{attribute 'qualified_only' := ''}
{attribute 'strict' := ''}
TYPE eFirmerVendorEvent2 :
(
	eNoInfo := 0,
	ePowerLimitationForHighTemperature := 1,
	ePowerLimitationForHighDCVoltage := 2,
	ePowerLimitationFromCapabilityRating := 3
);
END_TYPE

(* stored: Version 1.1.0.1, ProductVersion 3.1.4024.11
   DUT eFirmerVendorEvent2: Id {05b6aca2-57de-46dc-8a7d-71805fb1f0b4} *)
